TYPE ST_TCShuttlePOC :
STRUCT
	
		stGblParam: ST_TCSeqParam;
		fbTCShuttlePOCSeq: FB_TCShuttlePOCSeq;

END_STRUCT
END_TYPE

(* stored: Version 1.1.0.1, ProductVersion 3.1.4022.10
   DUT ST_TCShuttlePOC: Id {69db336d-75da-453e-9df1-c2c81184775b} *)
